FUNCTION_BLOCK Motor_Partida_Direta_HMI (* Service Interface Function Block Type *)
  (* Standard: 61499-2 *)
  (* Version 0.0, 15/01/2026, Schneider Electric, template *)
  PACKAGE Hidryco.HidrycoLib;
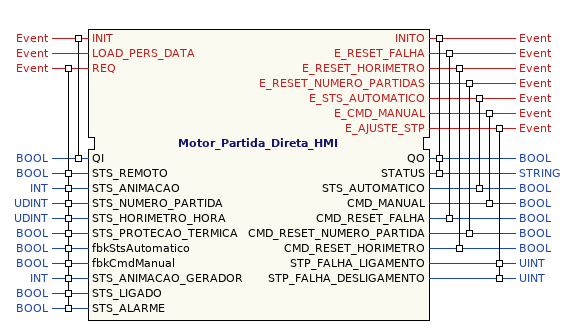
  EVENT_INPUT
    INIT WITH QI;
    LOAD_PERS_DATA;
    REQ WITH STS_REMOTO, STS_ANIMACAO, STS_NUMERO_PARTIDA, STS_HORIMETRO_HORA, fbkStsAutomatico, fbkCmdManual, STS_PROTECAO_TERMICA, STS_ANIMACAO_GERADOR, STS_LIGADO, STS_ALARME;
  END_EVENT
  EVENT_OUTPUT
    INITO WITH QO, STATUS;
    E_RESET_FALHA WITH CMD_RESET_FALHA;
    E_RESET_HORIMETRO WITH CMD_RESET_HORIMETRO;
    E_RESET_NUMERO_PARTIDAS WITH CMD_RESET_NUMERO_PARTIDA;
    E_STS_AUTOMATICO WITH STS_AUTOMATICO;
    E_CMD_MANUAL WITH CMD_MANUAL;
    E_AJUSTE_STP WITH STP_FALHA_LIGAMENTO, STP_FALHA_DESLIGAMENTO;
  END_EVENT
  VAR_INPUT
    QI : BOOL;
    STS_REMOTO : BOOL;
    STS_ANIMACAO : INT;
    STS_NUMERO_PARTIDA : UDINT;
    STS_HORIMETRO_HORA : UDINT;
    STS_PROTECAO_TERMICA : BOOL;
    fbkStsAutomatico : BOOL;
    fbkCmdManual : BOOL;
    STS_ANIMACAO_GERADOR : INT;
    STS_LIGADO : BOOL;
    STS_ALARME : BOOL;
  END_VAR
  VAR_OUTPUT
    QO : BOOL; (* Event Output Qualifier *)
    STATUS : STRING; (* Service Status *)
    STS_AUTOMATICO : BOOL;
    CMD_MANUAL : BOOL;
    CMD_RESET_FALHA : BOOL;
    CMD_RESET_NUMERO_PARTIDA : BOOL;
    CMD_RESET_HORIMETRO : BOOL;
    STP_FALHA_LIGAMENTO : UINT;
    STP_FALHA_DESLIGAMENTO : UINT;
  END_VAR
  SERVICE /
    SEQUENCE 
    END_SEQUENCE
  END_SERVICE
END_FUNCTION_BLOCK
